Staubli VAL3: velOverwrite.pgx

public program velOverwrite(bool x_bOverwriteVel)
begin

  // display velocity overwrite status

  if(x_bOverwriteVel == true)
    userPageSet("uxMonitor", "lblVelocityOverwrite", "innerHTML", "enabled")
  else
    userPageSet("uxMonitor", "lblVelocityOverwrite", "innerHTML", "disabled")
  endIf

end
